RoboDK station: CW2_M01044738_PDE4431.rdk

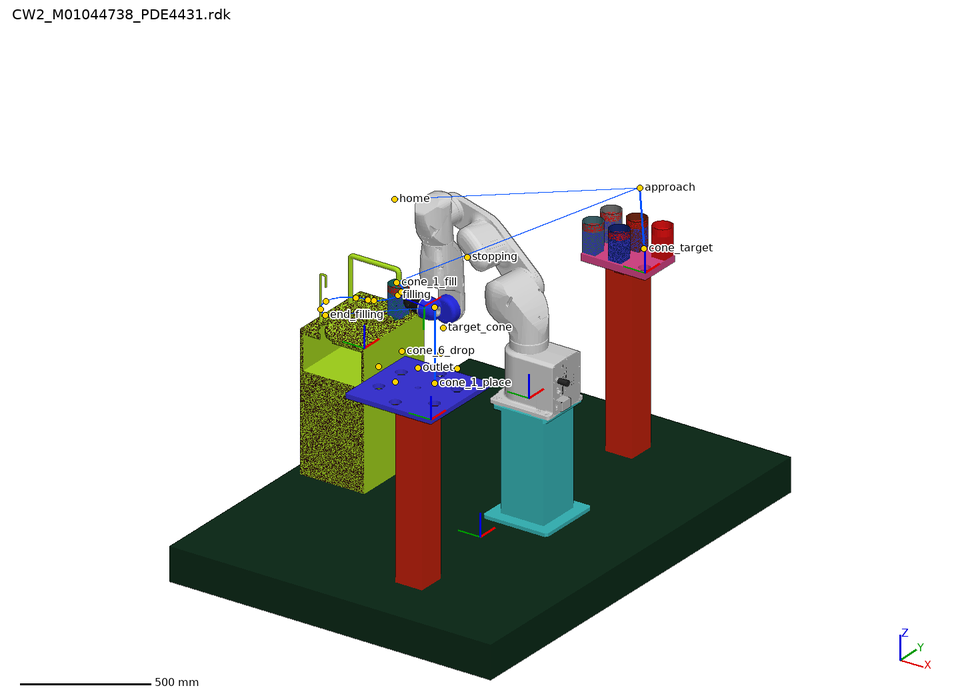
[picture v0: the station drawn from its stored meshes, robots at their saved joint values, targets as dots, program paths as lines]
Station PDE4431_CW2 (saved by RoboDK 5.8.0). Poses are relative to the parent item; angles as X-Y-Z fixed-axis rotations.
  - frame base_frame at (0, 0, 10) mm, rotated rx 0 ry 0 rz 90 deg
    - object PDE4431_CW2_2024 at (0, 0, 0) mm, rotated rx 90 ry 0 rz 0 deg, size 2000 x 980 x 1500 mm, geometry from PDE4431_CW2_2024.STEP
    - object Pedestal_3 at (38, -240, 150) mm, rotated rx 90 ry 0 rz 0 deg, size 300 x 480 x 300 mm, geometry from Pedestal_3.STEP
    - frame Epson VT6 Base at (40, -200, 630) mm
      - robot Epson VT6: 6 axes, payload 6 kg, reach 920 mm, repeatability 0.1 mm, weight 40 kg
          modified DH rows (alpha deg, a mm, theta deg, d mm): 0, 0, 0, 412; -90, 100, -90, 0; 0, 420, 0, 0; -90, 0, 0, 400; 90, 0, 0, 0; -90, 0, 0, 80
          base shift (0, 0, 0) mm, rotated rx 0 ry 0 rz 90 deg
          joint limits [-170, -160, -51, -200, -125, -360] to [170, 65, 190, 200, 125, 360]; home [0, 0, 0, 0, 0, 0]; saved at [-5.474, -59.896, -32.763, 0.959, 94.557, 0.375]
        - frame RobotiQ 2F-85 Gripper (Mechanism) Base at (0, 0, 0) mm, rotated rx 0 ry 0 rz 90 deg
          - robot RobotiQ 2F-85 Gripper (Mechanism) (model RobotiQ 2F85): 1 axes, payload 5 kg
              joint limits [0] to [85]; home [85]; saved at [60]
          - object cone_1 at (1.24, 29.98, 128.58) mm, rotated rx 75.54 ry -87.95 rz 104.81 deg, size 84.9 x 182 x 85 mm, geometry from Cone-Part.STEP
        - tool Tool 1, TCP at (0, 0, 130) mm
      - target gripper_open (Cartesian target) at (0, 683.92, 832) mm, rotated rx -90 ry 0 rz 0 deg; joints [85, 0, 0, 0, 0, 0] of RobotiQ 2F-85 Gripper (Mechanism)
      - target gripper_close (Cartesian target) at (0, 683.92, 832) mm, rotated rx -90 ry 0 rz 0 deg; joints [60, 0, 0, 0, 0, 0] of RobotiQ 2F-85 Gripper (Mechanism)
    - frame station_1_frame at (600, -350, 980) mm
      - target home (Cartesian target) at (-608.8, 742.44, 350) mm, rotated rx 19.99 ry -88.06 rz -110.51 deg; joints [1.443, 8.858, -28.234, -5.378, 21.283, 5.738] of Epson VT6
      - target cone_target (Cartesian target) at (40.44, 31.41, 80) mm, rotated rx 9.95 ry -88.07 rz 169.53 deg; joints [-105.167, -26.118, -40.115, 15.72, 68.941, -5.939] of Epson VT6
      - target approach (Cartesian target) at (10.44, 31.41, 350) mm, rotated rx 9.95 ry -88.07 rz 169.53 deg; joints [-105.201, 4.053, -24.07, 34.987, 26.23, -32.285] of Epson VT6
      - target cone_1_fill (Cartesian target) at (-408.8, 872.44, -119.95) mm, rotated rx 16 ry -88.06 rz -110.51 deg; joints [-18.802, -60.922, -18.262, 14.458, 81.382, -2.153] of Epson VT6
      - target filling (Cartesian target) at (-501.04, 802, -119.95) mm, rotated rx 9.87 ry -88.07 rz -104.39 deg; joints [-10.546, -59.86, -31.979, 6.038, 93.729, 0.524] of Epson VT6
      - target middle_fill (Cartesian target) at (-598.8, 872.44, -119.95) mm, rotated rx 16 ry -88.06 rz -107 deg; joints [0.272, -60.26, -22.861, -1.267, 84.985, 0.686] of Epson VT6
      - target middle_2_fill (Cartesian target) at (-698.8, 1000, -119.95) mm, rotated rx 9.99 ry -88.06 rz -100.51 deg; joints [8.938, -65.388, -0.069, -10.216, 67.714, 4.563] of Epson VT6
      - target end_filling (Cartesian target) at (-798.8, 932.44, -119.95) mm, rotated rx 16 ry -88.06 rz -107 deg; joints [19.47, -63.29, -7.421, -21.334, 73.82, 7.44] of Epson VT6
      - target cone_1_place (Cartesian target) at (-1375, 18, 74.97) mm, rotated rx 30.01 ry -88.07 rz -30.53 deg; joints [103.327, -36.989, -18.254, -16.365, 58.039, 10.213] of Epson VT6
      - target cone_1_retract (Cartesian target) at (-1375, 18, 400) mm, rotated rx 30.01 ry -88.07 rz -30.53 deg; joints [103.327, -12.172, 0.827, -47.435, 18.939, 47.222] of Epson VT6
      - target target_cone (Cartesian target) at (-1337.42, 3.34, 300.08) mm, rotated rx 39.89 ry -88.07 rz -30.41 deg; joints [101.8, -15.291, -10.13, -5.083, 26.998, 5.831] of Epson VT6
      - target cone_start (Cartesian target) at (-468.8, 808, -119.95) mm, rotated rx 16 ry -88.06 rz -110.51 deg; joints [-14.34, -59.806, -30.169, 9.838, 91.838, 0.53] of Epson VT6
      - target cone_station_1 (Cartesian target) at (-590, 852, -119.95) mm, rotated rx 9.87 ry -88.07 rz -104.39 deg; joints [0.759, -59.995, -25.833, -5.278, 87.745, 0.714] of Epson VT6
      - target cone_middle (Cartesian target) at (-608.8, 922.44, -119.95) mm, rotated rx 9.99 ry -88.06 rz -110.51 deg; joints [4.755, -61.742, -14.063, -15.596, 78.219, 4.118] of Epson VT6
      - target filling_station (Cartesian target) at (-768.8, 975, -119.95) mm, rotated rx 9.99 ry -88.06 rz -110.51 deg; joints [18.508, -65.639, 0.754, -31.046, 70.074, 12.988] of Epson VT6
      - target outlet (Cartesian target) at (-1301, 148, 74.97) mm, rotated rx 30.01 ry -88.07 rz -30.53 deg; joints [90.451, -30.034, -33.078, -1.06, 64.789, 1.446] of Epson VT6
      - target cone_2_drop (Cartesian target) at (-1451, 148, 74.97) mm, rotated rx 30.01 ry -88.07 rz -30.53 deg; joints [90.345, -42.143, -7.448, -1.095, 51.268, 1.676] of Epson VT6
      - target cone_3_drop (Cartesian target) at (-1377, 278, 74.97) mm, rotated rx 30.01 ry -88.07 rz -30.53 deg; joints [77.46, -37.007, -18.216, 14.262, 57.748, -7.115] of Epson VT6
      - target cone_4_drop (Cartesian target) at (-1225, 18, 79) mm, rotated rx 30.01 ry -88.07 rz -30.53 deg; joints [107.874, -25.434, -41.647, -19.605, 69.969, 8.477] of Epson VT6
      - target cone_6_drop (Cartesian target) at (-1225, 278, 78) mm, rotated rx 30.01 ry -88.07 rz -30.53 deg; joints [73.098, -25.439, -42.006, 17.463, 70.07, -5.646] of Epson VT6
      - target cone_5_drop (Cartesian target) at (-1151, 148, 78) mm, rotated rx 30.01 ry -88.07 rz -30.53 deg; joints [90.581, -19.834, -49.891, -1.149, 71.4, 1.364] of Epson VT6
      - target stopping (Cartesian target) at (-594.66, 411.86, 189.81) mm, rotated rx 179.62 ry 2.18 rz 87.53 deg; joints [7.54, 32.79, -35, 0, -90, -10] of Epson VT6
      - object cone_6 at (160, 270, 50) mm, rotated rx 90 ry 0 rz 0 deg, size 84.9 x 182 x 85 mm, geometry from Cone-Part.STEP
      - object cone_3 at (40, 270, 50) mm, rotated rx 90 ry 0 rz 0 deg, size 84.9 x 182 x 85 mm, geometry from Cone-Part.STEP
      - object cone_5 at (160, 150, 50) mm, rotated rx 90 ry 0 rz 0 deg, size 84.9 x 182 x 85 mm, geometry from Cone-Part.STEP
      - object cone_4 at (160, 30, 50) mm, rotated rx 90 ry 0 rz 0 deg, size 84.9 x 182 x 85 mm, geometry from Cone-Part.STEP
      - object cone_2 at (40, 150, 50) mm, rotated rx 90 ry 0 rz 0 deg, size 84.9 x 182 x 85 mm, geometry from Cone-Part.STEP
    - frame outlet_frame at (-900, -400, 970) mm
    - frame station_2_frame at (-200, 400, 770) mm
  - program gripper_open (2 instructions, listed below)
  - program gripper_close (2 instructions, listed below)
  - program program_1 (20 instructions, listed below)
  - program Replace (1 instructions, listed below)
  - Python program cone_station (listed below)
  - program AttachObject1 (1 instructions, listed below)
  - program DeattachObject1 (1 instructions, listed below)
  - Python program main_1 (listed below)
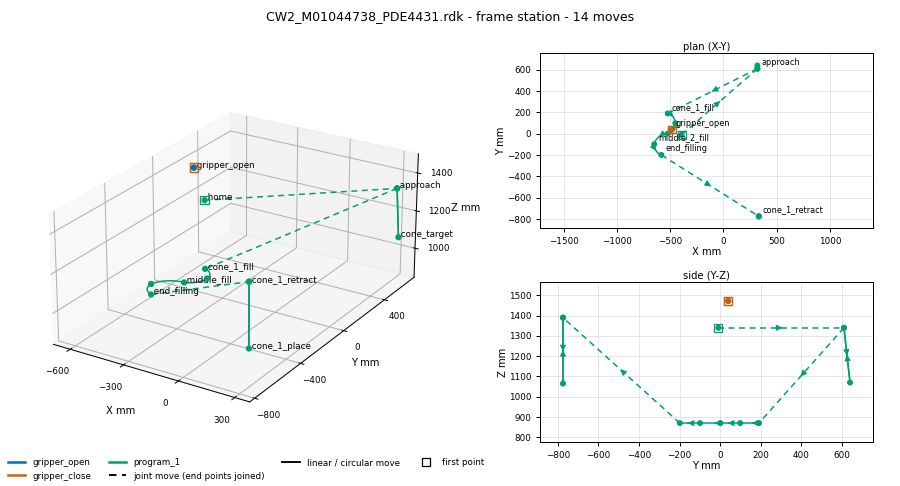
[picture p0: tool path of CW2_M01044738_PDE4431.rdk in frame station, 14 of 14 moves have a stored position in this frame; points joined in program order, loops and branches not executed]

--- program gripper_open (robot RobotiQ 2F-85 Gripper (Mechanism)) ---
  Set Ref.: Epson VT6 Base
  MoveJ (gripper_open)

--- program gripper_close (robot RobotiQ 2F-85 Gripper (Mechanism)) ---
  Set Ref.: Epson VT6 Base
  MoveJ (gripper_close)

--- program program_1 (robot Epson VT6) ---
  MoveJ (home)
  MoveJ (approach)
  Call gripper_open
  Set Ref.: station_1_frame
  Set Tool: Tool 1
  MoveL (cone_target)
  Call gripper_close
  Attach to Tool 1
  MoveL (approach)
  MoveJ (cone_1_fill)
  MoveC (cone_start, filling)
  MoveC (cone_station_1, middle_fill)
  MoveC (cone_middle, middle_2_fill)
  MoveC (filling_station, end_filling)
  MoveJ (cone_1_retract)
  MoveL (cone_1_place)
  Call gripper_open
  Detach from Tool 1
  MoveL (cone_1_retract)
  Set speed (500.0 mm/s)

--- program Replace (robot Epson VT6) ---
  Replace objects

--- Python program cone_station ---
from robodk.robolink import *  # Import the RoboDK API
from robodk.robomath import *  # Import RoboDK math utilities
import time

# Establish the connection with RoboDK
RDK = Robolink()

# Configure the robot and frames
robot_1 = RDK.Item('Epson VT6')  # Select the robot by name
station_1_frame = RDK.Item('station_1_frame')  # Initial frame for the object
outlet_frame = RDK.Item('outlet_frame')  # Final frame for the object

# Validate robot
if not robot_1.Valid():
    print("Error: Robot not found or invalid item")
    quit()

# Configure targets
home = RDK.Item('home')
approach = RDK.Item('approach')
cone_target = RDK.Item('cone_target')

# Validate targets
if not all([home.Valid(), approach.Valid(), cone_target.Valid()]):
    print("Error: One or more targets (home, approach, cone_target) are not valid")
    quit()

# Filling frame targets
filling_start = RDK.Item('cone_1_fill')
filling_cone_start = RDK.Item('cone_start')
filling_station_1 = RDK.Item('filling')
filling_cone_station_1 = RDK.Item('cone_station')
filling_middle = RDK.Item('middle_fill')
filling_cone_middle = RDK.Item('cone_middle')
filling_station_2 = RDK.Item('middle_2_fill')
filling_cone_station_2 = RDK.Item('filling_station')
filling_end = RDK.Item('end_filling')

# Outlet frame targets
retract_point = RDK.Item('cone_1_retract')
place_point = RDK.Item('cone_1_place')

# Validate outlet targets
if not all([retract_point.Valid(), place_point.Valid()]):
    print("Error: One or more outlet targets (cone_1_retract, cone_1_place) are not valid")
    quit()

# Gripper programs
gripper_open = RDK.Item('gripper_open', ITEM_TYPE_PROGRAM)
gripper_close = RDK.Item('gripper_close', ITEM_TYPE_PROGRAM)

# Validate gripper programs
if not gripper_open.Valid() or not gripper_close.Valid():
    print("Error: Gripper programs not found or invalid")
    quit()

# Object to attach
object_to_attach = RDK.Item('cone_1')

# Tool attachment
tool = robot_1.Childs()[0] if robot_1.Childs() else None

# Validate the tool and object
if not object_to_attach.Valid() or not tool.Valid():
    print("Error: Object or tool is not valid")
    quit()

print("Object and Tool set successfully.")

# Function to attach object to the tool
def TCP_On():
    """Attach the object to the robot's tool."""
    current_pose = object_to_attach.PoseAbs()
    object_to_attach.setParent(tool)
    object_to_attach.setPoseAbs(current_pose)
    print("Object attached to the tool.")

# Function to detach object from the tool
def TCP_Off():
    """Detach the object from the robot's tool and reattach it to the outlet frame."""
    current_pose = object_to_attach.PoseAbs()
    object_to_attach.setParent(outlet_frame)
    object_to_attach.setPoseAbs(current_pose)
    print("Object detached from the tool and reattached to the outlet frame.")

# Main sequence
def main():
    # Set the robot speed
    robot_1.setSpeed(50)

    # Move to the home position
    robot_1.MoveJ(home)

    # Pick the cone
    robot_1.MoveJ(approach)
    gripper_open.RunCode()
    time.sleep(0.5)
    robot_1.MoveL(cone_target)
    gripper_close.RunCode()
    TCP_On()
    time.sleep(0.5)
    robot_1.MoveL(approach)

    # Filling process
    robot_1.MoveJ(filling_start)
    robot_1.MoveC(filling_cone_start, filling_station_1)
    time.sleep(1)
    robot_1.MoveC(filling_cone_station_1, filling_middle)
    robot_1.MoveC(filling_cone_middle, filling_station_2)
    time.sleep(1)
    robot_1.MoveC(filling_cone_station_2, filling_end)

    # Place the cone
    robot_1.MoveJ(cone_1_retract)
    robot_1.MoveL(cone_1_place)
    gripper_open.RunCode()
    time.sleep(0.5)
    TCP_Off()
    time.sleep(0.5)
    robot_1.MoveL(cone_1_retract)

    # Return to home position
    robot_1.MoveJ(home)
    print("Task completed successfully.")

# Run the main sequence
main()

--- program AttachObject1 (robot Epson VT6) ---
  Attach to Tool 1

--- program DeattachObject1 (robot Epson VT6) ---
  Detach from Tool 1

--- Python program main_1 ---
from robodk.robolink import *  # Import the RoboDK API
from robodk.robomath import transl, rotz
from math import radians, cos, sin, atan2  # Use the standard math module
import time
import math

# Establishing the connection with RoboDK Robot
RDK = Robolink()  # Correctly instantiate the RoboDK connection

# Configuring two different robots as RoboDK items
robot_1 = RDK.Item('Epson VT6')  # Select the robot by name
station_1_frame = RDK.Item('station_1_frame')    # Initial frame of the object
outlet_frame = RDK.Item('outlet_frame')# Final frame for the object


if not robot_1.Valid():
    print("Error: Robot not found or invalid item")
    quit()

# Select the home target
home = RDK.Item('home')
#Feed frame Section
cone_approach = RDK.Item('approach')
cone_target = RDK.Item('cone_target')

cone1App_pos = RDK.Item("cone_approach")
secondApp_target =  cone1App_pos.Pose()*transl(0, -120, 0)
thirdApp_target =  cone1App_pos.Pose()*transl(0, -240, 0)
fourthApp_target =  cone1App_pos.Pose()*transl(0, 0, 120)
fifthApp_target =  cone1App_pos.Pose()*transl(0, -120, 120)
sixthApp_target =  cone1App_pos.Pose()*transl(0, -240, 120)

approachPoints = [cone_approach, secondApp_target, thirdApp_target, fourthApp_target, fifthApp_target, sixthApp_target]

cone1_pos = RDK.Item("cone_target")
second_target =  cone1_pos.Pose()*transl(0, -120, 0)
third_target =  cone1_pos.Pose()*transl(0, -240, 0)
fourth_target =  cone1_pos.Pose()*transl(0, 0, 120)
fifth_target =  cone1_pos.Pose()*transl(0, -120, 120)
sixth_target =  cone1_pos.Pose()*transl(0, -240, 120)

targetPoints = [cone_target, second_target, third_target, fourth_target, fifth_target, sixth_target]

cone_names = [
    'cone_1','cone_2','cone_3','cone_4','cone_5','cone_6',
]

#Filling frame Section

filling_start = RDK.Item('cone_1_fill')
filling_cone_start = RDK.Item('cone_start')
filling_station_1 = RDK.Item('filling')
filling_cone_station_1 = RDK.Item('cone_station')
filling_middle = RDK.Item('middle_fill')
filling_cone_middle = RDK.Item('cone_middle')
filling_station_2 = RDK.Item('middle_2_fill')
filling_cone_station_2 = RDK.Item('filling_station')
filling_end = RDK.Item('end_filling')

hexagonCenter = RDK.Item('centerOfOutlet_')  #hexagon center

#Outlet frame Section
cone1_filling_retract = RDK.Item('cone_1_retract')
cone2_RetractPoint = RDK.Item("cone2DropPoint").Pose()*transl(325.027, 0, 0)
cone3_RetractPoint = RDK.Item("cone3DropPoint").Pose()*transl(325.027, 0, 0)
cone4_RetractPoint = RDK.Item("cone4DropPoint").Pose()*transl(325.027, 0, 0)
cone5_RetractPoint = RDK.Item("cone5DropPoint").Pose()*transl(325.027, 0, 0)
cone6_RetractPoint = RDK.Item("cone6DropPoint").Pose()*transl(325.027, 0, 0)

cone_1_place = RDK.Item('cone_1_place')
cone2DropPoint = RDK.Item('cone_2_drop')
cone3DropPoint = RDK.Item('cone_3_drop')
cone4DropPoint = RDK.Item('cone_4_drop')
cone5DropPoint = RDK.Item('cone_5_drop')
cone6DropPoint = RDK.Item('cone_6_drop')

stopPoint = RDK.Item('stopping')

outlet_retractPoint = [cone_1_place, cone2_RetractPoint, cone3_RetractPoint, cone4_RetractPoint, cone5_RetractPoint, cone6_RetractPoint]
outlet_targetPoint = [cone_1_place, cone2DropPoint, cone3DropPoint, cone4DropPoint, cone5DropPoint, cone6DropPoint]


# Run a Python script program
gripper_open = RDK.Item('gripper_open', ITEM_TYPE_PROGRAM)  # For gripper open
gripper_close = RDK.Item('gripper_close', ITEM_TYPE_PROGRAM)  # For gripper close
Replace = RDK.Item('Replace_Corns', ITEM_TYPE_PROGRAM)  # For Cones back to feed frame


# Find the object to attach
object_to_attach = RDK.Item('cone_1')  # Replace 'Cone' with the name of your object

# Attach the object to the robot's tool
tool = robot_1.Childs()[0]  # Get the robot's tool (or specify the tool name directly)

if object_to_attach.Valid() and tool.Valid():
    print("Object and Tool set successfully.")
else:
    print("Error: Object and/or Tool is not valid.")

def TCP_On(object_to_attach):
    object_to_attach = RDK.Item(object_to_attach)
    current_pose = object_to_attach.PoseAbs()
    object_to_attach.setParent(tool)
    object_to_attach.setPoseAbs(current_pose)
    print("Object attached to the tool.")

def TCP_Off(object_to_attach):
    object_to_attach = RDK.Item(object_to_attach)
    current_pose = object_to_attach.PoseAbs()
    object_to_attach.setParent(outlet_frame)
    object_to_attach.setPoseAbs(current_pose)
    print("Object detached from the tool and reattached to Outlet Frame.")

def main():
    Replace.RunCode()
    robot_1.MoveJ(home)

    for n in range(6):
        # n = 1
        # Set the speed of the robot
        robot_1.setSpeed(100)  # Use the method on the robot item

        robot_1.MoveJ(approachPoints[n])
        gripper_open.RunCode()
        time.sleep(0.5)
        robot_1.MoveL(targetPoints[n])
        gripper_close.RunCode()
        time.sleep(1)
        TCP_On(cone_names[n])
        time.sleep(1)
        robot_1.MoveL(approachPoints[n])
        robot_1.MoveJ(filling_start)
        robot_1.MoveC(filling_cone_start, filling_station_1)
        time.sleep(1)
        robot_1.MoveC(filling_cone_station_1, filling_middle)
        robot_1.MoveC(filling_cone_middle, filling_station_2)
        time.sleep(1)
        robot_1.MoveC(filling_cone_station_2, filling_end)
        robot_1.MoveJ(outlet_retractPoint[n])
        robot_1.MoveL(outlet_targetPoint[n])
        gripper_open.RunCode()
        time.sleep(0.5)
        TCP_Off(cone_names[n])
        time.sleep(0.5)
        robot_1.MoveL(outlet_retractPoint[n])
        robot_1.MoveJ(home)

    robot_1.MoveJ(stopPoint)

main()
